FUNCTION_BLOCK Q_FontAttributes (* Command change font attributes ( Part 6 - F.28 ) *)
  (* Standard: ISO 11783-6; Description: Copyright (c) 2022 HR Agrartechnik GmbH This program and the accompanying materials are made available under the terms of the Eclipse Public License 2.0 which is available at https://www.eclipse.org/legal/epl-2.0/ SPDX-License-Identifier: EPL-2.0 see Description Tab *)
  (* Version 1.0, 2022-07-08, Franz Höpfinger, HR Agrartechnik GmbH *)
  PACKAGE isobus::ut;
  (* Documentation:
  Command change font attributes ( Part 6 - F.28 )
   This command is used to change the font attributes in a font attributes object.
   param[in] {objectID, uint16_t}
   Object ID
   param[in] {colour, uint8_t}
   New font colour (see Part 6 - A.3)
   param[in] {size, uint8_t}
   New font size (see Part 6 - B.14)
   param[in] {type, uint8_t}
   New font type (see Part 6 - B.14)
   param[in] {styleBitfield, uint8_t}
   New font style (see Part 6 - B.14)
   Return Values: 
   int16_t
    - VT_E_NO_ERR (0) - OK
   - VT_E_OVERFLOW (-6) - buffer overflow
   - VT_E_NOACT (-8) - Command not possible in current state
   - VT_E_NO_INSTANCE (-21) - No VT client available
   - VT_E_ISO_INSTANCE_INVALID (-129) - Identifier for instance (connection) invalid
   - VT_E_NOT_ALIVE (-130) - Identifier for instance valid, but VT Dead.
  *)
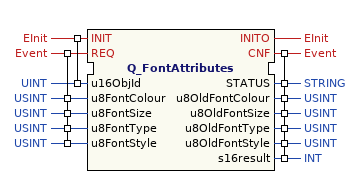
  EVENT_INPUT
    INIT : EInit WITH u16ObjId; (* Service Initialization *)
    REQ WITH u8FontColour, u8FontSize, u8FontType, u8FontStyle; (* Service Request *)
  END_EVENT
  EVENT_OUTPUT
    INITO : EInit; (* Initialization Confirm *)
    CNF WITH STATUS, u8OldFontType, u8OldFontColour, u8OldFontSize, s16result, u8OldFontStyle; (* Confirmation of Requested Service *)
  END_EVENT
  VAR_INPUT
    u16ObjId : UINT; (* Object ID *)
    u8FontColour : USINT; (* New font colour (see Part 6 - A.3) *)
    u8FontSize : USINT; (* New font size (see Part 6 - B.14) *)
    u8FontType : USINT; (* New font type (see Part 6 - B.14) *)
    u8FontStyle : USINT; (* New font style (see Part 6 - B.14) *)
  END_VAR
  VAR_OUTPUT
    STATUS : STRING; (* Service Status *)
    u8OldFontColour : USINT; (* Old font colour (see Part 6 - A.3) *)
    u8OldFontSize : USINT; (* Old font size (see Part 6 - B.14) *)
    u8OldFontType : USINT; (* Old font type (see Part 6 - B.14) *)
    u8OldFontStyle : USINT; (* Old font style (see Part 6 - B.14) *)
    s16result : INT; (* retval see description *)
  END_VAR
END_FUNCTION_BLOCK
